VAR_GLOBAL CONSTANT
	cusiMinAddedChilds: USINT := 1;
END_VAR

(* stored: Version 1.1.0.1, ProductVersion 3.1.0.19
   GVL Const_SLB: Id {db30b4f5-61af-4ec4-bf1c-7741c7d85d0f} *)
